FUNCTION_BLOCK FB_Alarms
VAR_INPUT
END_VAR
VAR_OUTPUT
END_VAR
VAR
END_VAR

METHOD M_IntializeAlarms
VAR_INPUT
END_VAR
END_METHOD

END_FUNCTION_BLOCK

(* stored: Version 1.1.0.1, ProductVersion 3.1.4024.9
   POU FB_Alarms: Id {d2513749-01b3-4d38-a6bd-fec59f5b66e3}, SpecialFunc None
   Method M_IntializeAlarms: Id {ee998365-2dc3-4348-b184-4d2a49cea2fe} *)
